FUNCTION_BLOCK FB_QuenchTank
VAR_INPUT
	sAction 				: STRING(10);			// 'fill', 'drain'
END_VAR

VAR_OUTPUT
	bError					: BOOL;
	nWaterTemp				: USINT;				// scaled value of thermocouple
	sErrorMsg				: STRING(60);
END_VAR

VAR
	tDrainTimeout           : TIME := T#10S;		// time until drain is aborted
	tFillTimeout			: TIME := T#10S;		// time until fill is aborted
	tPumpEnableDelay		: TIME := T#3S;			// delay to allow drain valve to open before pump is enabled
	tmrFillTimer			: Tc2_Standard.TON;
	tmrDrainTimer			: Tc2_Standard.TON;
END_VAR

IF sAction = 'fill' THEN
	tmrFillTimer(IN := TRUE, PT := tFillTimeout);
	IF NOT tmrFillTimer.Q THEN
		GVL.boOpenFillValve := TRUE;
		bError := FALSE;
		sErrorMsg := '';
	ELSE
		GVL.boOpenFillValve := FALSE;
		bError := TRUE;
		sErrorMsg := 'Timeout while filling tank - check float high level sensor';
	END_IF

ELSIF sAction = 'drain' THEN
	tmrDrainTimer(IN := TRUE, PT := tDrainTimeout);
	GVL.boOpenDrainValve := TRUE;
	IF tmrDrainTimer.ET > tPumpEnableDelay THEN
		GVL.boEnablePump := TRUE;
	END_IF
ELSE
	tmrDrainTimer(IN := FALSE);
	tmrFillTimer(IN := FALSE);
END_IF

METHOD M_DrainTank : BOOL
VAR_INPUT
END_VAR
END_METHOD

METHOD M_FillTank : BOOL
VAR_INPUT
END_VAR
END_METHOD

END_FUNCTION_BLOCK

(* stored: Version 1.1.0.1, ProductVersion 3.1.4024.11
   POU FB_QuenchTank: Id {a0e2e726-f3b1-46e4-a948-9b07cbe723bb}, SpecialFunc None
   Method M_DrainTank: Id {f2311ade-b7b2-4b22-8411-9cb761205599}
   Method M_FillTank: Id {7fce20e2-fe8f-455d-92d6-51ae4650f517} *)
